// TwinCAT 3 PLC project Library
// Title: lcls-twincat-motion-sheppard
// Company: SLAC
// ProjectVersion: 0.0.0
// ProgramVersion: 3.1.4020.5
// libraries:
//   Tc2_EtherCAT, * (Beckhoff Automation GmbH)
//   Tc2_MC2, * (Beckhoff Automation GmbH)
//   Tc2_Standard, * (Beckhoff Automation GmbH)
//   Tc2_System, * (Beckhoff Automation GmbH)
//   Tc2_Utilities, * (Beckhoff Automation GmbH)
//   TcUnit, * (www.tcunit.org)
// project tree:
//   DUTs/ DUT_MotionStage.TcDUT, EL5042_Status.TcDUT (not stored), ENUM_EpicsHomeCmd.TcDUT (not stored), ENUM_EpicsMotorCmd.TcDUT (not stored), ENUM_StageBrakeMode.TcDUT (not stored), ENUM_StageEnableMode.TcDUT (not stored), ST_RenishawAbsEnc.TcDUT (not stored)
//   POUs/Motion/ FB_GantryDiffVirtualLimitSwitch.TcPOU (not stored), FB_MotionStage.TcPOU
//   POUs/Testing/ FB_MicroStepCountTest.TcPOU (not stored)
//   tc_mca_std_lib/DUTs/ DUT_AxisStatus_v0_01.TcDUT (not stored)
//   tc_mca_std_lib/GVLs/ GVL.TcGVL (not stored)
//   tc_mca_std_lib/POUs/ChangeConfig/ FB_ReadFloatParameter.TcPOU (not stored), FB_ReadParameterInNc_v1_00.TcPOU (not stored), FB_WriteFloatParameter.TcPOU (not stored), FB_WriteParameterInNc_v1_00.TcPOU (not stored)
//   tc_mca_std_lib/POUs/ErrorHandling/ DUT_ErrorState.TcDUT (not stored), DUT_TerminalError.TcDUT (not stored), FB_ErrorList.TcPOU (not stored), FB_TerminalError.TcPOU (not stored), GVL_ErrorSystem.TcGVL (not stored), ST_ErrorSystem.TcDUT (not stored)
//   tc_mca_std_lib/POUs/Hardware/EtherCAT_Terminals/Analog_Inputs/ EL3174_0002.TcPOU (not stored), EL3214.TcPOU (not stored), EL3255.TcPOU (not stored), FB_CalculateFrequency_3702_v0_01.TcPOU (not stored)
//   tc_mca_std_lib/POUs/Hardware/EtherCAT_Terminals/Digital_Inputs/ EL1008.TcPOU (not stored), EL1018.TcPOU (not stored), EL1808.TcPOU (not stored), EL1809.TcPOU (not stored), EL1819.TcPOU (not stored), FB_EL1252ASM_v1_00.TcPOU (not stored)
//   tc_mca_std_lib/POUs/Hardware/EtherCAT_Terminals/Digital_Outputs/ EL2014.TcPOU (not stored), EL2252.TcPOU (not stored), EL2808.TcPOU (not stored), EL2819.TcPOU (not stored)
//   tc_mca_std_lib/POUs/Hardware/EtherCAT_Terminals/Digital_Outputs/External_Types/ dutEL2521_Ctrl.TcDUT (not stored), dutEL2521_Status.TcDUT (not stored)
//   tc_mca_std_lib/POUs/Hardware/EtherCAT_Terminals/Measuring_Terminals/ EL5002.TcPOU (not stored), EL5021.TcPOU (not stored), EL5042.TcPOU (not stored), EL5101.TcPOU (not stored)
//   tc_mca_std_lib/POUs/Hardware/EtherCAT_Terminals/Motion/ EL7211_v1_00.TcPOU (not stored), EL9576_v1_00.TcPOU (not stored)
//   tc_mca_std_lib/POUs/Hardware/EtherCAT_Terminals/System/ EL9410.TcPOU (not stored), EL9505.TcPOU (not stored)
//   tc_mca_std_lib/POUs/Hardware/Other/ EK1200.TcPOU (not stored)
//   tc_mca_std_lib/POUs/Motion/ FB_DriveVirtual.TcPOU (not stored), FB_NcAxis.TcPOU (not stored)
//   tc_mca_std_lib/POUs/Motion/Homing/ FB_HomeDirect.TcPOU (not stored), FB_HomeFinish.TcPOU (not stored), FB_HomePrepare.TcPOU (not stored), FB_HomeReadNcVelocities.TcPOU (not stored), FB_HomeReadSoftLimEnable.TcPOU (not stored), FB_HomeToSwitch.TcPOU (not stored), FB_HomeVirtual.TcPOU (not stored), FB_HomeWriteNcVelocities.TcPOU (not stored), FB_HomeWriteSoftLimEnable.TcPOU (not stored)
//   Version/ Global_Version.TcGVL

// ---- DUTs/DUT_MotionStage.TcDUT
TYPE DUT_MotionStage :
STRUCT
	// Hardware
	Axis: AXIS_REF;
	{attribute 'pytmc' := '
		pv: LimitForwardEnable
		io: i
	'}
	bLimitForwardEnable AT %I*: BOOL;
	{attribute 'pytmc' := '
		pv: LimitBackwardEnable
		io: i
	'}
	bLimitBackwardEnable AT %I*: BOOL;
	bHome AT %I*: BOOL;

	bBrakeRelease AT %Q*: BOOL;
	
	// Psuedo-hardware
	{attribute 'pytmc' := '
		pv: AllForwardEnable
		io: i
	'}
	bAllForwardEnable: BOOL:=FALSE; // Forward enable EPS summary
	{attribute 'pytmc' := '
		pv: AllBackwardEnable
		io: i
	'}
	bAllBackwardEnable: BOOL:=FALSE; // Forward enable EPS summary
	bHardwareEnable AT %I*: BOOL; // True when Emergency stop button is not activated
	{attribute 'pytmc' := '
		pv: AllEnable
		io: i
	'}
	bAllEnable: BOOL:=FALSE; // Enable EPS summary encapsulating emergency stop button and any additional motion preventive hardware

	{attribute 'pytmc' := '
		pv: GantryForwardEnable
		io: i
	'}
	bGantryForwardEnable: BOOL:=FALSE; // Forward virtual gantry limit switch
	{attribute 'pytmc' := '
		pv: GantryBackwardEnable
		io: i
	'}
	bGantryBackwardEnable: BOOL:=FALSE; // Reverse virtual gantry limit switch
	
	// Settings
	bPowerSelf: BOOL:=TRUE;
	{attribute 'pytmc' := '
		pv: EnableMode
		io: o
	'}
	nEnableMode: INT:=ENUM_StageEnableMode.STAGE_ENABLE_MOTION;
	nBrakeMode: INT:=ENUM_StageBrakeMode.STAGE_BRAKE_DISABLED;
	nHomingMode: INT:=ENUM_EpicsHomeCmd.EPICS_MOTOR_HOME_NONE;
	
	bGantryAxis: BOOL:=FALSE; // Set true to activate gantry EPS
	nGantryTol: LINT:=0; // Set to gantry difference tolerance
	nEncRef: ULINT:=0; // Encoder count at which this axis is aligned with other axis
	
	// Commands
	{attribute 'pytmc' := '
		pv: Enable
		io: o
	'}
	bEnable: BOOL;
	bReset: BOOL;
	bExecute: BOOL;
	
	// Args
	nCommand: INT;
	nCmdData: INT;
	fPosition: LREAL;
	fVelocity: LREAL;
	fAcceleration: LREAL;
	fDeceleration: LREAL;
	fHomePosition: LREAL;
	
	// Info
	nMotionAxisID: UDINT:=0;
	
	// Returns
	{attribute 'pytmc' := '
		pv: EnableDone
		io: i
	'}
	bEnableDone: BOOL;
	bBusy: BOOL;
	bDone: BOOL;
	bError: BOOL;
	sErrorMessage: STRING;
	stAxisStatus: DUT_AxisStatus_v0_01;
END_STRUCT
END_TYPE

// ---- Version/Global_Version.TcGVL
{attribute 'TcGenerated'}
// This function has been automatically generated from the project information.
VAR_GLOBAL CONSTANT
	{attribute 'const_non_replaced'}
	{attribute 'linkalways'}
	stLibVersion_lcls_twincat_motion_sheppard : ST_LibVersion := (iMajor := 0, iMinor := 0, iBuild := 0, iRevision := 0, sVersion := '0.0.0');
END_VAR

// ---- POUs/Motion/FB_MotionStage.TcPOU
FUNCTION_BLOCK FB_MotionStage
VAR_IN_OUT
	stMotionStage: DUT_MotionStage;
END_VAR
VAR
	fbDriveVirtual: FB_DriveVirtual;
	bExecute: BOOL;
	bFwdHit: BOOL;
	bBwdHit: BOOL;
	fbExecFallingEdge: F_TRIG;
	bIsCoupled : BOOL;
END_VAR

// Start with an accurate status
stMotionStage.Axis.ReadStatus();

// Handle auto-enable timing
CASE stMotionStage.nEnableMode OF
	ENUM_StageEnableMode.STAGE_ENABLE_ALWAYS:
		stMotionStage.bEnable := TRUE;
		bExecute := stMotionStage.bExecute;
	ENUM_StageEnableMode.STAGE_ENABLE_NEVER:
		bExecute := stMotionStage.bExecute;
	ENUM_StageEnableMode.STAGE_ENABLE_MOTION:
		IF stMotionStage.bExecute THEN
			stMotionStage.bEnable := TRUE;
		END_IF
		bExecute := stMotionStage.bExecute AND stMotionStage.bEnabled;
END_CASE

// Automatically fill the correct nCmdData for homing
IF stMotionStage.nCommand = ENUM_EpicsMotorCmd.EPICS_MOTOR_HOME THEN
	stMotionStage.nCmdData := stMotionStage.nHomingMode;
END_IF

// EPS Directional Enables
stMotionStage.bLimAllFwd := stMotionStage.bLimFwd AND (stMotionStage.bLimGntFwd OR NOT stMotionStage.bGantryAxis);
stMotionStage.bLimAllBwd := stMotionStage.bLimBwd AND (stMotionStage.bLimGntBwd OR NOT stMotionStage.bGantryAxis);

// Handle standard commands using ESS's FB
fbDriveVirtual(En:=TRUE,
	bEnable:=stMotionStage.bEnable AND stMotionStage.bSTO,
	bReset:=stMotionStage.bReset,
	bExecute:=bExecute,
	nCommand:=INT_TO_UINT(stMotionStage.nCommand),
	nCmdData:=INT_TO_UINT(stMotionStage.nCmdData),
	fVelocity:=stMotionStage.fVelocity,
	fPosition:=stMotionStage.fPosition,
	fAcceleration:=stMotionStage.fAcceleration,
	fDeceleration:=stMotionStage.fDeceleration,
	bLimitFwd:=stMotionStage.bLimAllFwd,
	bLimitBwd:=stMotionStage.bLimAllBwd,
	bHomeSensor:=stMotionStage.bHome,
	fHomePosition:=stMotionStage.fHomePosition,
	bPowerSelf:=stMotionStage.bPowerSelf,
	nMotionAxisID=>stMotionStage.nMotionAxisID,
	bError=>stMotionStage.bError,
	sErrorMessage=>stMotionStage.sErrorMessage,
	Axis:=stMotionStage.Axis);

IF fbDriveVirtual.bBusy THEN
	stMotionStage.bBusy := TRUE;
	stMotionStage.bDone := FALSE;
END_IF

IF stMotionStage.bError THEN
	stMotionStage.bBusy := FALSE;
	stMotionStage.bDone := FALSE;
	stMotionStage.bEnable := FALSE;
END_IF

// Check the limits and cancel execution if appropriate. Without this block we have infinite error spam
bFwdHit := stMotionStage.Axis.Status.PositiveDirection AND NOT stMotionStage.bLimAllFwd;
bBwdHit := stMotionStage.Axis.Status.NegativeDirection AND NOT stMotionStage.bLimAllBwd;
IF bFwdHit OR bBwdHit THEN
	stMotionStage.bExecute := FALSE;
END_IF

// Mark done if settled or if unexpected stop, then reset the FB if there is no error
fbExecFallingEdge(CLK:=stMotionStage.bExecute);
IF (stMotionStage.Axis.Status.InTargetPosition AND NOT fbDriveVirtual.bBusy) OR fbExecFallingEdge.Q THEN
	IF NOT stMotionStage.bDone THEN
		stMotionStage.bDone := TRUE;
		stMotionStage.bBusy := FALSE;
		IF NOT stMotionStage.Axis.Status.Error THEN
			bExecute := FALSE;
			stMotionStage.bExecute := FALSE;
		END_IF
	END_IF
END_IF
IF stMotionStage.nEnableMode = ENUM_StageEnableMode.STAGE_ENABLE_MOTION AND NOT bExecute THEN
	IF stMotionStage.Axis.Status.MotionState = MC_AXISSTATE_STANDSTILL THEN
		stMotionStage.bEnable := FALSE;
	END_IF
END_IF

// Get a definitive bEnabled reading
CASE stMotionStage.Axis.Status.MotionState OF
	// We are not enabled if there is an issue
	MC_AXISSTATE_UNDEFINED, MC_AXISSTATE_DISABLED, MC_AXISSTATE_ERRORSTOP:
		stMotionStage.bEnabled := FALSE;
	ELSE
		stMotionStage.bEnabled := TRUE;
END_CASE

// Handle the brake. TRUE means brake disabled.
CASE stMotionStage.nBrakeMode OF
	ENUM_StageBrakeMode.STAGE_BRAKE_DISABLED:
		stMotionStage.bBrake := stMotionStage.bEnabled AND stMotionStage.bExecute;
	ENUM_StageBrakeMode.STAGE_BRAKE_STANDSTILL:
		IF stMotionStage.Axis.Status.MotionState = MC_AXISSTATE_STANDSTILL THEN
			stMotionStage.bBrake := FALSE;
		ELSE
			stMotionStage.bBrake := TRUE;
		END_IF
END_CASE
CASE stMotionStage.Axis.Status.MotionState OF
	MC_AXISSTATE_UNDEFINED, MC_AXISSTATE_ERRORSTOP:
		stMotionStage.bBrake := FALSE;
END_CASE

// Sync the epics status struct
stMotionStage.stAxisStatus := fbDriveVirtual.stAxisStatus;
stMotionStage.stAxisStatus.bEnabled := stMotionStage.bEnabled;

// Reset everything when bReset is flagged
IF stMotionStage.bReset THEN
	stMotionStage.bEnable := FALSE;
	stMotionStage.bReset := FALSE;
	stMotionStage.bExecute := FALSE;
	bExecute := FALSE;
END_IF

// Ignore homing if we have the setting for it
// e.g. for pre-calibrated absolute encoders
IF stMotionStage.nHomingMode = ENUM_EpicsHomeCmd.EPICS_MOTOR_HOME_NONE THEN
	stMotionStage.stAxisStatus.bHomed := TRUE;
END_IF

END_FUNCTION_BLOCK
